VAR_GLOBAL
	Prg				: FB_Program(0);
END_VAR

(* stored: Version 1.1.0.1
   GVL GVL_Program: Id {88f81564-0663-4c0a-bef0-b24c283c5d6c} *)
